FUNCTION_BLOCK FB_System_Test EXTENDS TcUnit.FB_TestSuite
VAR
	fbSystem : FB_System;
END_VAR

TestInitialization();
TestProperties();

METHOD TestInitialization
VAR
	fbGetCurTaskIdx 	: TC2_SYSTEM.GETCURTASKINDEX;
	fResult 	: REAL;
	fExpected 	: REAL;
	bResult 	: BOOL;
	bExpected 	: BOOL;
END_VAR
TEST('Before InitRun fTimeScaling is 0');
fExpected := 0;
fResult := fbSystem.fTimeScaling;
AssertEquals(Expected := fExpected,
             Actual := fResult,
             Message := 'Result value is not correct');
TEST_FINISHED();

TEST('Before InitRun fDeltaTime is 0');
fExpected := 0;
fResult := fbSystem.fDeltaTime;
AssertEquals(Expected := fExpected,
             Actual := fResult,
             Message := 'Result value is not correct');	
TEST_FINISHED();

TEST('Before InitRun GVL_IOSEF.refSystem is NULL');
bExpected := FALSE;
bResult := __ISVALIDREF(GVL_Core.refSystem);
AssertEquals(Expected := bExpected,
             Actual := bResult,
             Message := 'Result value is not correct');	
TEST_FINISHED();

fbSystem();

TEST('After InitRun fTimeScaling > 0');
fExpected := 1;
fResult := fbSystem.fTimeScaling;
AssertEquals(Expected := fExpected,
             Actual := fResult,
             Message := 'Result value is not correct');
TEST_FINISHED();

TEST('After InitRun fDeltaTime > 0');
fbGetCurTaskIdx();
fExpected := UDINT_TO_REAL(TwinCAT_SystemInfoVarList._TaskInfo[fbGetCurTaskIdx.index].CycleTime / 10000) / 1000.0;
fResult := fbSystem.fDeltaTime;
AssertEquals(Expected := fExpected,
             Actual := fResult,
             Message := 'Result value is not correct');	
TEST_FINISHED();

TEST('After InitRun GVL_IOSEF.refSystem is Valid');
bExpected := TRUE;
bResult := __ISVALIDREF(GVL_Core.refSystem);
AssertEquals(Expected := bExpected,
             Actual := bResult,
             Message := 'Result value is not correct');	
TEST_FINISHED();
END_METHOD

METHOD TestProperties : REFERENCE TO FB_Test
VAR
	fbGetCurTaskIdx 	: TC2_SYSTEM.GETCURTASKINDEX;
	fResult 	: REAL;
	fExpected 	: REAL;
END_VAR
TEST('Test Property: bDebug');
fbSystem.bDebug := TRUE;
AssertTRUE(Condition := fbSystem.bDebug,  Message := 'Property value is not correct');	
TEST_FINISHED();

TEST('Test Property: bVerbose');
fbSystem.bVerbose := TRUE;
AssertTRUE(Condition := fbSystem.bVerbose,  Message := 'Property value is not correct');	
TEST_FINISHED();

TEST('Test Property: fTimeScaling Initial');
fExpected := 1;
fResult := fbSystem.fTimeScaling;
AssertEquals(Expected := fExpected,
             Actual := fResult,
             Message := 'Result value is not correct');
TEST_FINISHED();

TEST('Test Property: fTimeScaling Zero');
fbSystem.fTimeScaling := 0;
fExpected := 1;
fResult := fbSystem.fTimeScaling;
AssertEquals(Expected := fExpected,
             Actual := fResult,
             Message := 'Result value is not correct');
TEST_FINISHED();

TEST('Test Property: fTimeScaling Limit Min');
fbSystem.fTimeScaling := -1;
fExpected := 0.01000001;
fResult := fbSystem.fTimeScaling;
AssertEquals(Expected := fExpected,
             Actual := fResult,
             Message := 'Result value is not correct');
TEST_FINISHED();

TEST('Test Property: fTimeScaling Limit Max');
fbSystem.fTimeScaling := 1E+6;
fExpected := 100;
fResult := fbSystem.fTimeScaling;
AssertEquals(Expected := fExpected,
             Actual := fResult,
             Message := 'Result value is not correct');
TEST_FINISHED();

TEST('Test Property: fTimeScaling In Range_1');
fbSystem.fTimeScaling := 2;
fExpected := 2;
fResult := fbSystem.fTimeScaling;
AssertEquals(Expected := fExpected,
             Actual := fResult,
             Message := 'Result value is not correct');
TEST_FINISHED();

TEST('Test Property: fTimeScaling In Range_2');
fbSystem.fTimeScaling := 1;
fExpected := 1;
fResult := fbSystem.fTimeScaling;
AssertEquals(Expected := fExpected,
             Actual := fResult,
             Message := 'Result value is not correct');
TEST_FINISHED();
END_METHOD

END_FUNCTION_BLOCK

(* stored: Version 1.1.0.1, ProductVersion 3.1.4024.12
   POU FB_System_Test: Id {b63e147c-75bf-0bab-19ac-fcb11587783f}, SpecialFunc None
   Method TestInitialization: Id {770f9dc1-e523-003a-32ad-e3dd6b6e5f7f}
   Method TestProperties: Id {68ce1d1e-3fa5-08f7-1698-d31eaaaf1320} *)
